PROGRAM Main_Background
VAR
END_VAR

(* execute background processes *)
Background_Time();
//Background_IMU();
//Background_FatigueCam();
Background_GPS();

END_PROGRAM

(* stored: Version 1.1.0.1, ProductVersion 3.1.4024.6
   POU Main_Background: Id {bf39ed73-1e87-4530-9028-00e14babda15}, SpecialFunc None *)
